FUNCTION_BLOCK Multiplexer
  (* Standard: 61499-2 *)
  (* Version 0.2, 2003-12-04, JHC, Rockwell Automation, Renamed for better indexing. *)
  (* Version 0.1, 2002-11-05, JHC, Rockwell Automation, Corrected missing ST element in Algorithm REQ. *)
  (* Version 0.0, 2000-05-30, JHC, Rockwell Automation *)
  (* Compiler header: package fb.rt.benchmarks.watermonitor; *)
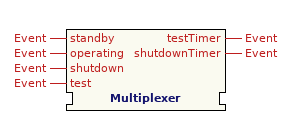
  EVENT_INPUT
    standby;
    operating;
    shutdown;
    test;
  END_EVENT
  EVENT_OUTPUT
    testTimer; (* system has gone in/out of TEST mode *)
    shutdownTimer; (* system has gone in/out of SHUTDOWN mode *)
  END_EVENT
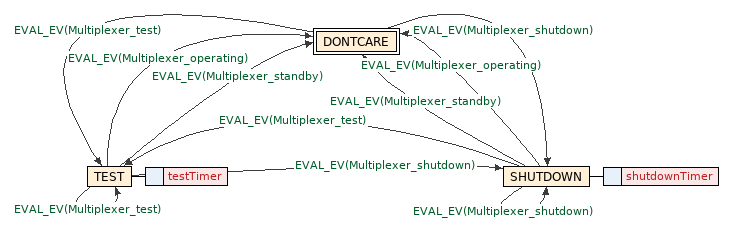
  EC_STATES
    DONTCARE;
    SHUTDOWN : -> shutdownTimer;
    TEST : -> testTimer; (* Normal execution *)
  END_STATES
  EC_TRANSITIONS
    DONTCARE TO TEST := EVAL_EV(Multiplexer_test);
    DONTCARE TO SHUTDOWN := EVAL_EV(Multiplexer_shutdown);
    TEST TO TEST := EVAL_EV(Multiplexer_test);
    TEST TO SHUTDOWN := EVAL_EV(Multiplexer_shutdown);
    TEST TO DONTCARE := EVAL_EV(Multiplexer_operating);
    TEST TO DONTCARE := EVAL_EV(Multiplexer_standby);
    SHUTDOWN TO SHUTDOWN := EVAL_EV(Multiplexer_shutdown);
    SHUTDOWN TO TEST := EVAL_EV(Multiplexer_test);
    SHUTDOWN TO DONTCARE := EVAL_EV(Multiplexer_operating);
    SHUTDOWN TO DONTCARE := EVAL_EV(Multiplexer_standby);
  END_TRANSITIONS
END_FUNCTION_BLOCK
